// TIA Portal project "AutomationHeatExchanger_2" (V14)

(* hardware
DEVICE "S7300/ET200M station_1"  S7-300 station
   slot 0: "Rail_0"  Rail  6ES7 390-1***0-0AA0
   slot 2: "PLC_1"  CPU 314C-2 PN/DP  6ES7 314-6EH04-0AB0  V3.3
      slot 2: "PROFINET interface_1"  PN-IO
         slot 1: "Port_1"  Port
         slot 2: "Port_2"  Port
      slot 5: "DI 24/DO 16_1"  DI24/DO16
      slot 6: "AI 5/AO 2_1"  AI5/AO2
      slot 7: "Count_1"  Counter
      slot 8: "Positioning_1"  Positioning
*)

// ===== PLC "PLC_1"  CPU 314C-2 PN/DP =====

DATA_BLOCK "Paras"   // DB1
{ S7_Optimized_Access := 'FALSE' }
VERSION : 0.1
   VAR
      Tenp_SP : Real := 120.0;   // Temp setpoint
      Temp_PV : Real;
      Power : Real;
      Kp : Real := -1.7;
      Ti : Time := T#78s;
      COM_RST : Bool;
      MAN_ON : Bool;
   END_VAR
BEGIN
END_DATA_BLOCK

DATA_BLOCK "Model_DB"   // DB2
{ S7_Optimized_Access := 'FALSE' }
VERSION : 0.1
// stored: InstanceOfName Model
"Model"
BEGIN
END_DATA_BLOCK

FUNCTION_BLOCK "Model"   // FB1, SCL
{ S7_Optimized_Access := 'FALSE' }
VERSION : 0.1
   VAR_INPUT
      CO : Real := 39.0;
   END_VAR
   VAR_OUTPUT
      PV : Real := 130.0;
   END_VAR
   VAR
      CO_Delay : Array[1..48] of Real;
      PV1 : Real := 140.0;
      index : Int := 1;
   END_VAR
BEGIN
   IF #index <= 48 THEN
       #CO_Delay[#index] := #CO;
   ELSE
       #PV := 0.987 * #PV1 - 0.006929 * #CO_Delay[#index-48] + 2.048;
       #PV1 := #PV;
       #CO_Delay[#index - 48] := #CO;
       IF ((#index - 48) >= 48) THEN
           #index := 48;
       END_IF;
   END_IF;
   #index := #index + 1;
END_FUNCTION_BLOCK

ORGANIZATION_BLOCK "Main"   // OB1, LAD
TITLE = "Main Program Sweep (Cycle)"
{ S7_Optimized_Access := 'FALSE' }
VERSION : 0.1
   VAR_TEMP
      OB1_EV_CLASS : Byte;   // Bits 0-3 = 1 (Coming event), Bits 4-7 = 1 (Event class 1)
      OB1_SCAN_1 : Byte;   // 1 (Cold restart scan 1 of OB 1), 3 (Scan 2-n of OB 1)
      OB1_PRIORITY : Byte;   // Priority of OB Execution
      OB1_OB_NUMBR : Byte;   // 1 (Organization block 1, OB1)
      OB1_RESERVED_1 : Byte;   // Reserved for system
      OB1_RESERVED_2 : Byte;   // Reserved for system
      OB1_PREV_CYCLE : Int;   // Cycle time of previous OB1 scan (milliseconds)
      OB1_MIN_CYCLE : Int;   // Minimum cycle time of OB1 (milliseconds)
      OB1_MAX_CYCLE : Int;   // Maximum cycle time of OB1 (milliseconds)
      OB1_DATE_TIME : Date_And_Time;   // Date and time OB1 started
   END_VAR
BEGIN
END_ORGANIZATION_BLOCK

ORGANIZATION_BLOCK "CYC_INT2"   // OB32, FBD
TITLE = "Cyclic Interrupt"
{ S7_Optimized_Access := 'FALSE' }
VERSION : 0.1
   VAR_TEMP
      OB32_EV_CLASS : Byte;   // Bits 0-3 = 1 (Coming event), Bits 4-7 = 1 (Event class 1)
      OB32_STRT_INF : Byte;   // 16#33 (OB 32 has started)
      OB32_PRIORITY : Byte;   // Priority of OB Execution
      OB32_OB_NUMBR : Byte;   // 32 (Organization block 32, OB32)
      OB32_RESERVED_1 : Byte;   // Reserved for system
      OB32_RESERVED_2 : Byte;   // Reserved for system
      OB32_PHS_OFFSET : Int;   // Phase offset (integer, milliseconds)
      OB32_RESERVED_3 : Int;   // Reserved for system
      OB32_EXC_FREQ : Int;   // Frequency of execution (msec)
      OB32_DATE_TIME : Date_And_Time;   // Date and time OB32 started
   END_VAR
BEGIN

REGION Network 1
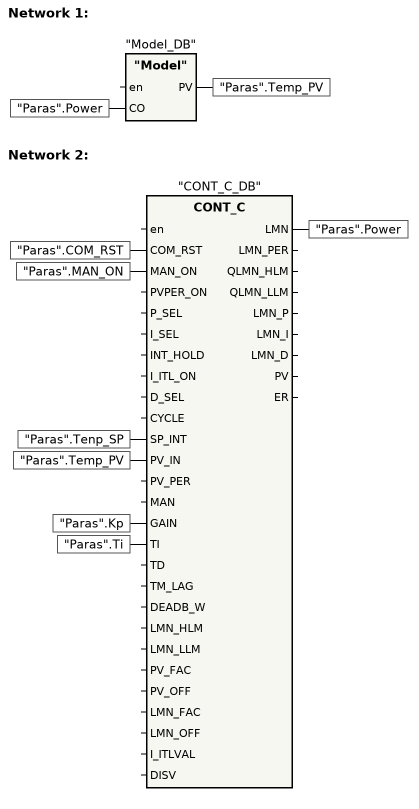
   "Model_DB"(CO := "Paras".Power, PV => "Paras".Temp_PV);   // "Model"
END_REGION

REGION Network 2
   "CONT_C_DB"(COM_RST := "Paras".COM_RST,   // CONT_C
               MAN_ON := "Paras".MAN_ON,
               SP_INT := "Paras".Tenp_SP,
               PV_IN := "Paras".Temp_PV,
               GAIN := "Paras".Kp,
               TI := "Paras".Ti,
               LMN => "Paras".Power);
END_REGION
END_ORGANIZATION_BLOCK